{attribute 'qualified_only'}
VAR_GLOBAL
	// Pitch Mechanism:
	{attribute 'TcLinkTo' := '.diEncCnt:=TIIB[EL5042_M1_PitchBender]^FB Inputs Channel 1^Position'}
	MR2L3_Pitch : HOMS_PitchMechanism := (ReqPosLimHi := 220,
		                                 ReqPosLimLo := -193.0,
		                                 diEncPosLimHi := 11216281,
		                                 diEncPosLimLo := 11004512);
END_VAR

(* stored: Version 1.1.0.1, ProductVersion 3.1.4022.18
   GVL GVL_MR2L3: Id {39aa3d3e-e981-4a44-9c10-e2ef2b749839} *)
